FUNCTION_BLOCK FB_StationTakeLoad
VAR_INPUT
	Enable:				BOOL;
	System:				REFERENCE TO ST_System;
	Station:			REFERENCE TO ST_SystemStation;
	Error:				REFERENCE TO ST_Error;
	Setting:			REFERENCE TO ST_Setting;
	Recipe:				REFERENCE TO ST_Recipe;	
	Parameter:			REFERENCE TO ST_StationTakeLoad;
END_VAR
VAR_OUTPUT
END_VAR
VAR
	_i:					INT;
	_arrTon:		    ARRAY[0..20] OF TON;
	_arrFbErrorTag:		ARRAY[0..20] OF FB_ErrorTag;
	_arrState:			ARRAY[0..20] OF BOOL;
	
	_iMoveAbsIndex1:	UINT;
	_iMoveAbsIndex2:	UINT;
	_bIsZWork:			BOOL;// 取Line0为真 其他情况为假
	_stHandshake: ST_StationTakeLoadHandshake;
END_VAR

A_Auto();
A_Home();

ACTION A_Auto:
CASE Station.iStepNow OF
	1000:
		Station.arrInfo[E_Language.Chinese]:="初始化完成 等待启动";
		IF Enable THEN
			Station.iStepNext:=1101;
		END_IF
	1101:
		Station.arrInfo[E_Language.Chinese]:="取料信号判断";
		Parameter.eState:=E_StationState.Load;
		Setting.eTakeModeBuffer:=E_TakeMode.None;
		Station.iStepNext:=1111;
	1111:
		IF Setting.eTakeModeBuffer=E_TakeMode.None THEN
			Setting.eTakeModeBuffer:=Setting.eTakeMode;
		ELSE
			Parameter.eState:=E_StationState.Busy;
			Station.iStepNext:=1151;
		END_IF
	1151:
		Station.arrInfo[E_Language.Chinese]:="请求取料";
		CASE Setting.eTakeModeBuffer OF
			E_TakeMode.Take0:
				_iMoveAbsIndex1:=2;
				_bIsZWork:=TRUE;
				Parameter.stHandshake.bRequestLine0Buffer_T0 :=TRUE;
				IF Parameter.stHandshake.bResponseTake_T0 THEN
					Station.iStepNext:=1201;
				END_IF
			E_TakeMode.Take1:
				_iMoveAbsIndex1:=3;
				_bIsZWork:=FALSE;
				Parameter.stHandshake.bRequestLineLoad_T1:=TRUE;
				IF Parameter.stHandshake.bResponseTake_T1 THEN
					Station.iStepNext:=1201;
				END_IF
			E_TakeMode.Take3Load:
				_iMoveAbsIndex1:=4;
				_bIsZWork:=FALSE;
				Parameter.stHandshake.bRequestLineLoad_T3:=TRUE;
				IF Parameter.stHandshake.bResponseTake_T3 THEN
					Station.iStepNext:=1201;
				END_IF
			E_TakeMode.None:
				Station.iStepNext:=1101;
		END_CASE
	1201:
		Station.arrInfo[E_Language.Chinese]:="Y轴至取料位";
		Parameter.eState:=E_StationState.Busy;
		IF Parameter.fbTakeY.M_MoveAbs(_iMoveAbsIndex1) THEN
			Station.iStepNext:=1301;
		END_IF
	1301:
		Station.arrInfo[E_Language.Chinese]:="Z模组下降";
		IF M_ZWork()  THEN
			Station.iStepNext:=1401;
		END_IF
	1401:
		Station.arrInfo[E_Language.Chinese]:="夹紧气缸夹紧";
		IF Parameter.fbTakeClamp.M_WorkRequest() THEN
			Station.iStepNext:=1501;
		END_IF
	1501:
		Station.arrInfo[E_Language.Chinese]:="Z模组上升";
		IF M_ZHome() THEN
			Station.iStepNext:=1511;
		END_IF
	1511:
		Station.arrInfo[E_Language.Chinese]:="复位取料请求 ";
		CASE Setting.eTakeModeBuffer OF
			E_TakeMode.Take0:
				Parameter.stHandshake.bRequestLine0Buffer_T0 :=FALSE;
				IF NOT Parameter.stHandshake.bResponseTake_T0 THEN
					Station.iStepNext:=1601;
				END_IF
			E_TakeMode.Take1:
				Parameter.stHandshake.bRequestLineLoad_T1:=FALSE;
				IF NOT Parameter.stHandshake.bResponseTake_T1 THEN
					Station.iStepNext:=1601;
				END_IF
			E_TakeMode.Take3Load:
				Parameter.stHandshake.bRequestLineLoad_T3:=FALSE;
				IF NOT Parameter.stHandshake.bResponseTake_T3 THEN
					Station.iStepNext:=1601;
				END_IF
		END_CASE
	1601:
		Station.arrInfo[E_Language.Chinese]:="请求放料";
		Parameter.eState:=E_StationState.Done;
		Setting.eTakeModeBuffer:=E_TakeMode.None;
		Station.iStepNext:=1611;
	1611:
		IF Setting.eTakeModeBuffer=E_TakeMode.None THEN
			Setting.eTakeModeBuffer:=Setting.eTakeMode;
		ELSE
			Parameter.eState:=E_StationState.Busy;
			Station.iStepNext:=1651;
		END_IF
	1651:
		_bIsZWork:=FALSE;
		CASE Setting.eTakeModeBuffer OF
			E_TakeMode.Place1:
				_iMoveAbsIndex2:=3;
				Parameter.stHandshake.bRequestLineLoad_P1:=TRUE;
				IF Parameter.stHandshake.bResponseTake_P1 THEN
					Station.iStepNext:=1701;
				END_IF
			E_TakeMode.Place3Load:
				_iMoveAbsIndex2:=4;
				Parameter.stHandshake.bRequestLineLoad_P3:=TRUE;
				IF Parameter.stHandshake.bResponseTake_P3 THEN
					Station.iStepNext:=1701;
				END_IF
		END_CASE
	1701:
		Station.arrInfo[E_Language.Chinese]:="等待Y轴至放料位";
		IF Parameter.fbTakeY.M_MoveAbs(_iMoveAbsIndex2) THEN
			Station.iStepNext:=1801;
		END_IF
	1801:
		Station.arrInfo[E_Language.Chinese]:="Z模组下降";
		IF M_ZWork() THEN
			Station.iStepNext:=1901;
		END_IF
	1901:
		Station.arrInfo[E_Language.Chinese]:="夹紧气缸松开";
		IF Parameter.fbTakeClamp.M_HomeRequest() THEN
			Station.iStepNext:=2001;
		END_IF
	2001:
		Station.arrInfo[E_Language.Chinese]:="Z模组上升";
		IF M_ZHome() THEN
			Station.iStepNext:=2101;
		END_IF
	2101:
		Station.arrInfo[E_Language.Chinese]:="复位放料请求";
		CASE Setting.eTakeModeBuffer OF
			E_TakeMode.Place1:
				Parameter.stHandshake.bRequestLineLoad_P1:=FALSE;
				IF NOT Parameter.stHandshake.bResponseTake_P1 THEN
					Station.iStepNext:=2201;
				END_IF
			E_TakeMode.Place3Load:
				Parameter.stHandshake.bRequestLineLoad_P3:=FALSE;
				IF NOT Parameter.stHandshake.bResponseTake_P3 THEN
					Station.iStepNext:=2201;
				END_IF
		END_CASE
	2201:
		Station.arrInfo[E_Language.Chinese]:="Y轴至初始位";
		IF Parameter.fbTakeY.M_MoveAbs(1) THEN
			Station.iStepNext:=1101;
		END_IF
END_CASE
END_ACTION

ACTION A_Home:
CASE Station.iStepNow OF
	0:
		Station.arrInfo[E_Language.Chinese]:="等待初始化";
		Parameter.stHandshake:=_stHandshake;
		Parameter.eState:=E_StationState.None;
		Setting.eTakeModeBuffer:=E_TakeMode.None;
		Station.iStepNext:=SEL(Enable,1000,500);
	500:
		Station.arrInfo[E_Language.Chinese]:="夹紧气缸松开";
		IF Parameter.fbTakeClamp.M_HomeRequest() THEN
			Station.iStepNext:=600;
		END_IF
	600:
		Station.arrInfo[E_Language.Chinese]:="Z模组初始化";
		IF M_ZInit() THEN
			Station.iStepNext:=700;
		END_IF
	700:
		Station.arrInfo[E_Language.Chinese]:="Z模组至上升位";
		IF M_ZHome() THEN
			Station.iStepNext:=800;
		END_IF
	800:
		Station.arrInfo[E_Language.Chinese]:="Y模组回零";
		IF Parameter.fbTakeY.M_Home() THEN
			Station.iStepNext:=900;
		END_IF
	900:
		Station.arrInfo[E_Language.Chinese]:="Y模组至初始位";
		IF Parameter.fbTakeY.M_MoveAbs(1) THEN
			Station.iStepNext:=1000;
		END_IF
END_CASE
END_ACTION

METHOD M_ZHome : BOOL
VAR_INPUT
END_VAR
CASE Recipe.eMachineType OF
	E_MachineType.LH311,E_MachineType.RH311:
		M_ZHome:=Parameter.fbTakeLift1.M_HomeRequest() AND Parameter.fbTakeLift2.M_HomeRequest();
	E_MachineType.LH353,E_MachineType.RH353:
		M_ZHome:=Parameter.fbTakeZ.M_MoveAbs(1);
	E_MachineType.LH367,E_MachineType.RH367:
		M_ZHome:=Parameter.fbTakeLift1.M_HomeRequest() AND Parameter.fbTakeLift2.M_HomeRequest();
	E_MachineType.LH201,E_MachineType.RH201:
		M_ZHome:=Parameter.fbTakeZ.M_MoveAbs(1);
	E_MachineType.LH069,E_MachineType.RH069:
		M_ZHome:=Parameter.fbTakeZ.M_MoveAbs(1);
	E_MachineType.LH373,E_MachineType.RH373:
		M_ZHome:=Parameter.fbTakeZ.M_MoveAbs(1);
END_CASE
END_METHOD

METHOD M_ZInit : BOOL
VAR_INPUT
END_VAR
CASE Recipe.eMachineType OF
	E_MachineType.LH311,E_MachineType.RH311:
		M_ZInit:=TRUE;
	E_MachineType.LH353,E_MachineType.RH353:
		M_ZInit:=Parameter.fbTakeZ.M_Home();
	E_MachineType.LH367,E_MachineType.RH367:
		M_ZInit:=TRUE;
	E_MachineType.LH201,E_MachineType.RH201:
		M_ZInit:=Parameter.fbTakeZ.M_Home();
	E_MachineType.LH069,E_MachineType.RH069:
		M_ZInit:=Parameter.fbTakeZ.M_Home();
	E_MachineType.LH373,E_MachineType.RH373:
		M_ZInit:=Parameter.fbTakeZ.M_Home();
END_CASE
END_METHOD

METHOD M_ZWork : BOOL
VAR_INPUT
END_VAR
CASE Recipe.eMachineType OF
	E_MachineType.LH311,E_MachineType.RH311:
		M_ZWork:=Parameter.fbTakeLift1.M_WorkRequest() AND Parameter.fbTakeLift2.M_WorkRequest();
	E_MachineType.LH353,E_MachineType.RH353:
		M_ZWork:=SEL(_bIsZWork,Parameter.fbTakeZ.M_MoveAbs(3) ,Parameter.fbTakeZ.M_MoveAbs(2));
	E_MachineType.LH367,E_MachineType.RH367:
		M_ZWork:=Parameter.fbTakeLift1.M_WorkRequest() AND SEL(_bIsZWork,TRUE ,Parameter.fbTakeLift2.M_WorkRequest()) ;
	E_MachineType.LH201,E_MachineType.RH201:
		M_ZWork:=SEL(_bIsZWork,Parameter.fbTakeZ.M_MoveAbs(3) ,Parameter.fbTakeZ.M_MoveAbs(2));
	E_MachineType.LH069,E_MachineType.RH069:
		M_ZWork:=SEL(_bIsZWork,Parameter.fbTakeZ.M_MoveAbs(3) ,Parameter.fbTakeZ.M_MoveAbs(2));
	E_MachineType.LH373,E_MachineType.RH373:
		M_ZWork:=SEL(_bIsZWork,Parameter.fbTakeZ.M_MoveAbs(3) ,Parameter.fbTakeZ.M_MoveAbs(2));
END_CASE
END_METHOD

END_FUNCTION_BLOCK

(* stored: Version 1.1.0.1, ProductVersion 3.1.4024.3
   POU FB_StationTakeLoad: Id {44e51563-5233-4a3b-af5c-f0758ecc2e44}, SpecialFunc None
   Action A_Auto: Id {e67ac0db-1360-4197-89c1-be0f8410c1c6}
   Action A_Home: Id {78e05fe3-7f8d-4689-bb0e-3db8190b8255}
   Method M_ZHome: Id {23ccd6e4-3dd2-420a-955f-6f2f01f3b9cf}
   Method M_ZInit: Id {1f4f8bd6-cd62-4dcf-aba0-594630fd9ffd}
   Method M_ZWork: Id {69eddb07-6a77-4cbf-a886-69bb012a7c39} *)
